FUNCTION_BLOCK PUBLIC FB_VAC_GEN
VAR_IN_OUT
	Hardware : TYP_VAC_GEN_HW;
END_VAR
VAR_INPUT
	Control : TYP_VAC_GEN_CTRL;
	Config : TYP_VAC_GEN_CONF;
	AlarmConfig : TYP_ALARM_DEVICE_CONFIG;
END_VAR
VAR_OUTPUT
	Status : TYP_VAC_GEN_STATUS;
END_VAR
VAR
	CmdActivate : BOOL;
	CmdRelease : BOOL;
	VacAlarm : FB_ALARM;
	VacAlarmTime : TON;
	VacAlarmEdge : R_TRIG;
	ServiceEdge : R_TRIG;
	ReleaseTime : TIME;
END_VAR

VacAlarm.Config.Acknowledge := E_ALARM_ACK_TYPE.ACK_AND_RESET;
VacAlarm.Config.Name := CONCAT(AlarmConfig.Name, '*NO_VAC');
VacAlarm(Handler := AlarmConfig.Handler);
VacAlarmTime(IN := CmdActivate AND NOT Status.ReachedVac, PT := Config.Alarm.Timeout);
VacAlarmEdge(CLK := VacAlarmTime.Q);

IF VacAlarmEdge.Q AND Config.Alarm.Enable THEN
	VacAlarm.Activate();
END_IF;

IF NOT CmdActivate AND VacAlarm.IsActive THEN
	VacAlarm.Reset();
END_IF;

ServiceEdge(CLK := Control.ServiceEnable);

IF ServiceEdge.Q THEN // Remember command when entering service mode to avoid unpredictable movements
	Control.ServiceActivate := CmdActivate;
	Control.ServiceRelease := CmdRelease;
END_IF;

IF Control.ServiceEnable THEN
	CmdActivate := Control.ServiceActivate;
	CmdRelease := Control.ServiceRelease;
END_IF;

Hardware.Out.EnableVac := CmdActivate;
Hardware.Out.ReleaseVac := CmdRelease;

Status.ReachedVac := Hardware.In.ReachedVac;
Status.Error := VacAlarm.IsActive;

IF NOT Control.ServiceEnable THEN
	IF Status.ReachedVac AND NOT Config.Permanent THEN
		Hardware.Out.EnableVac := FALSE;
	END_IF;
	
	IF CmdRelease AND TIME() - ReleaseTime > T#1S THEN
		CmdRelease := FALSE;
	END_IF;
END_IF;

METHOD PUBLIC Activate : REFERENCE TO FB_VAC_GEN
VAR_INPUT
END_VAR
IF THIS^.Control.Enable AND THIS^.Control.EnableActivate THEN
	CmdActivate := TRUE;
	CmdRelease := FALSE;
END_IF;

Activate REF= THIS^;
END_METHOD

METHOD PUBLIC Release : REFERENCE TO FB_VAC_GEN
VAR_INPUT
END_VAR
IF THIS^.Control.Enable AND THIS^.Control.EnableRelease THEN
	CmdActivate := FALSE;
	CmdRelease := TRUE;
	ReleaseTime := TIME();
END_IF;

Release REF= THIS^;
END_METHOD

METHOD PUBLIC Reset : REFERENCE TO FB_VAC_GEN
VAR_INPUT
END_VAR

CmdActivate := FALSE;
CmdRelease := FALSE;


Reset REF= THIS^;
END_METHOD

END_FUNCTION_BLOCK

(* stored: Version 1.1.0.1, ProductVersion 3.1.4024.12
   POU FB_VAC_GEN: Id {b1869338-79d5-4ea3-ac76-0e830783f544}, SpecialFunc None
   Method Activate: Id {d68b21ec-e267-49c3-86f3-e067eb1056b1}
   Method Release: Id {fe7bb3ce-673c-425c-8892-7a43e04fdf9a}
   Method Reset: Id {d7e120fa-93bd-42da-be10-337805f1d266} *)
